(*
:Author: Takashi Ichihashi
:Date: 2023-03-07

Decreration
=========================

.. code-block:: 

	// Variables for queue feature
	fb_deq : dequeue;
	get_data : T_Arg;
	// databuffer for 1 second with 10 ms time delta
    queue_buffer: ARRAY[0..99] OF T_Arg;
	

Useage
=================

This is example code that the sInputData is queued in and queued out for sOutputData.

.. code-block:: 

	// put_data
	IF NOT fb_deq.full THEN

		sInputData := ANY_DATA;
		// put pointer
		fb_deq.put(F_BIGTYPE(ADR(sInputData),SIZEOF(sInputData)));

	END_IF
	
	// getting data
	get_data := fb_deq.get();
	MEMCPY(ADR(sOutputData), get_data.pData, get_data.cbLen);
	
	
*)

FUNCTION_BLOCK dequeue
VAR
	_queue_usage:	UDINT;
	_queue_size:	UDINT := DbLibParam.COMMAND_QUEUE_BUFFER_SIZE;
	nWriteIndex: 	UDINT;
	nReadIndex: 	UDINT;
	queue_buffer:	ARRAY [0..DbLibParam.COMMAND_QUEUE_BUFFER_SIZE - 1] OF ChunkCommand;
END_VAR

PROPERTY full : BOOL
GET
full :=  _queue_usage >= DBLibParam.COMMAND_QUEUE_BUFFER_SIZE - 1;
END_GET
END_PROPERTY

METHOD get : ChunkCommand
VAR_INPUT
END_VAR
//Set buffer index

IF _queue_usage > 0 THEN
	get := queue_buffer[nReadIndex];
	get.accumulated_amount := get.accumulated_amount - get.chunk_size;
	_queue_usage := _queue_usage - 1;
	nReadIndex := nReadIndex + 1;
	IF nReadIndex > DBLibParam.COMMAND_QUEUE_BUFFER_SIZE - 1 THEN
		nReadIndex := 0;
	END_IF
END_IF

RETURN;
END_METHOD

PROPERTY PUBLIC index : UDINT
GET
index := nWriteIndex;
END_GET
END_PROPERTY

PROPERTY PUBLIC max_index : UDINT
GET
max_index := DBLibParam.COMMAND_QUEUE_BUFFER_SIZE - 1;
END_GET
END_PROPERTY

METHOD PUBLIC put : UDINT
VAR_INPUT
	lData:	ChunkCommand;
END_VAR
//Set buffer index

IF _queue_usage >= DBLibParam.COMMAND_QUEUE_BUFFER_SIZE - 1 THEN
	put := 0;
ELSE
	queue_buffer[nWriteIndex] := lData;
	lData.accumulated_amount := lData.accumulated_amount + lData.chunk_size;
	_queue_usage := _queue_usage + 1;
	nWriteIndex := nWriteIndex + 1;
	IF nWriteIndex > DBLibParam.COMMAND_QUEUE_BUFFER_SIZE - 1 THEN
		nWriteIndex := 0;
	END_IF
	put := 1;
END_IF

RETURN;
END_METHOD

PROPERTY queue_size : UDINT
GET
queue_size := _queue_size;
END_GET
END_PROPERTY

PROPERTY queue_usage : UDINT
GET
queue_usage := _queue_usage;
END_GET
END_PROPERTY

END_FUNCTION_BLOCK

(* stored: Version 1.1.0.1, ProductVersion 3.1.4024.12
   POU dequeue: Id {40b5d0f5-5c4a-4c21-b039-6567ed0f3ed3}, SpecialFunc None
   Property full: Id {2090bbfa-cf3b-42d9-83cb-c8801d1b5ffd}
   Get Get: Id {11d8a220-140d-44af-91dc-0c0b14043cba}
   Method get: Id {8b74c0af-e452-4b04-80b6-4bc8c107a41d}
   Property index: Id {797924aa-4aac-4502-9933-1db6ff110751}
   Get Get: Id {1aa0817d-5541-4bd9-8c6c-c4f73615a599}
   Property max_index: Id {d2cc1e4e-f8ed-4e95-bcc4-f73c95718a81}
   Get Get: Id {d83f4ff6-13c9-4c3f-9065-ce9aeb94ccfb}
   Method put: Id {bc495a1c-f6bd-4bba-8df0-e2c2c6cddb62}
   Property queue_size: Id {8ced692f-17fa-4590-b6bd-53841bf68804}
   Get Get: Id {dfdc89e1-eeb1-4141-9046-b5b43fa9d899}
   Property queue_usage: Id {6eb19352-bb31-4ae0-8d30-bb26bad7bb02}
   Get Get: Id {2d47a586-eb1f-401e-b5b0-233891fb8ef8} *)
